// TIA Portal V19 export
TYPE "UDT_COUNTER"
   STRUCT
      Trigger : Bool := false;
      Pulse : Bool := false;
      Reset : Bool := false;
      End : Bool := false;
      Target { S7_SetPoint := 'True'} : Int := 0;
      Actual : Int := 0;
      Remaining : Int := 0;
   END_STRUCT;
END_TYPE
